% RSLogix 500 project InventoryManagement.RSS, saved by version 8.30.00.16 %
PROJECT "UNTITLED"    % processor: Bul.1763 MicroLogix 1100 Series B %

PROGRAM FILES
  LAD 2   9 rungs

DATA FILES
  O0 OUTPUT  4 elements
  I1 INPUT  6 elements
  S2 STATUS  66 elements
  B3 BINARY  1 elements
  T4 TIMER  1 elements
  C5 COUNTER  1 elements
  R6 CONTROL  1 elements
  N7 INTEGER  11 elements
  F8 FLOAT  1 elements
  ST9 STRING  10 elements

LADDER 2
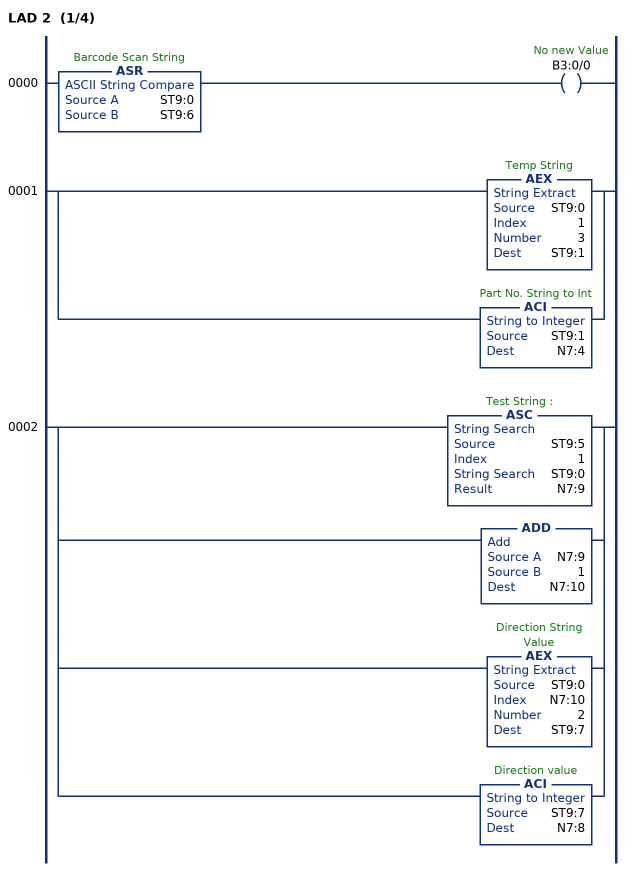
% Rung: 0 %
SOR ASR ST9:0 ST9:6 OTE B3:0/0 EOR
%   ST9:0  "Barcode Scan String" %
%   B3:0/0  "No new Value" %
% Rung: 1 %
SOR BST AEX ST9:0 1 3 ST9:1 NXB ACI ST9:1 N7:4 BND EOR
%   ST9:0  "Barcode Scan String" %
%   ST9:1  "Temp String" %
%   N7:4  "Part No. String to Int" %
% Rung: 2 %
SOR BST ASC ST9:5 1 ST9:0 N7:9 NXB ADD N7:9 1 N7:10 NXB AEX ST9:0 N7:10 2 ST9:7 NXB ACI ST9:7 N7:8 BND EOR
%   ST9:5  "Test String :" %
%   ST9:0  "Barcode Scan String" %
%   ST9:7  "Direction String Value" %
%   N7:8  "Direction value" %

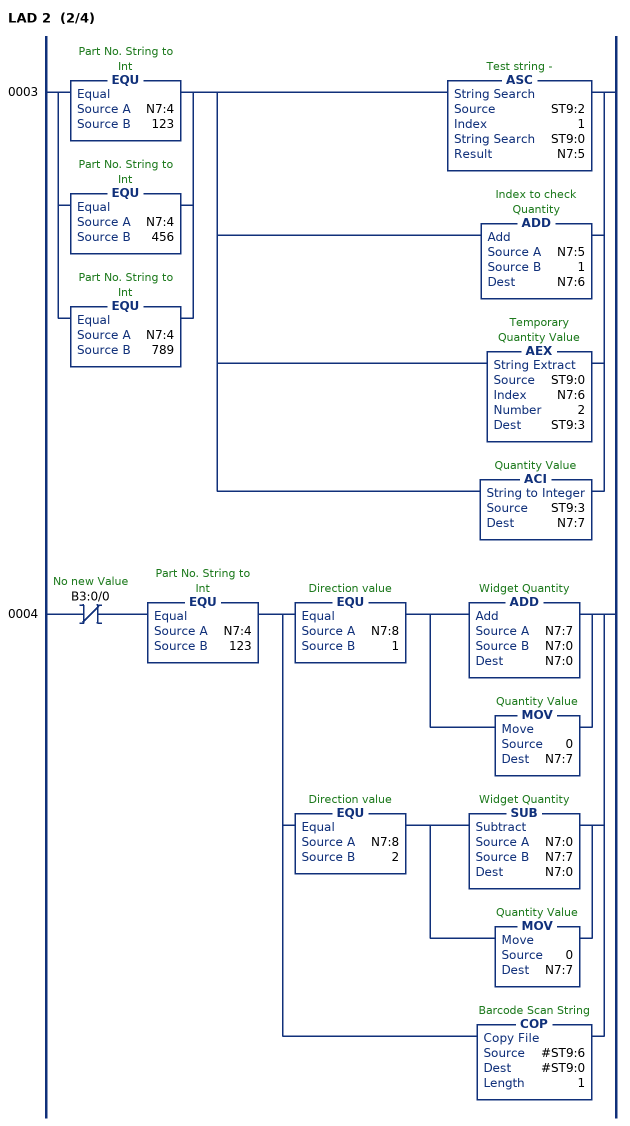
% Rung: 3 %
SOR BST EQU N7:4 123 NXB EQU N7:4 456 NXB EQU N7:4 789 BND BST ASC ST9:2 1 ST9:0 N7:5 NXB ADD N7:5 1 N7:6 NXB AEX ST9:0 N7:6 2 ST9:3 NXB ACI ST9:3 N7:7 BND EOR
%   N7:4  "Part No. String to Int" %
%   ST9:2  "Test string -" %
%   ST9:0  "Barcode Scan String" %
%   N7:5  "Target Start Index" %
%   N7:6  "Index to check Quantity" %
%   ST9:3  "Temporary Quantity Value" %
%   N7:7  "Quantity Value" %
% Rung: 4 %
SOR XIO B3:0/0 EQU N7:4 123 BST EQU N7:8 1 BST ADD N7:7 N7:0 N7:0 NXB MOV 0 N7:7 BND NXB EQU N7:8 2 BST SUB N7:0 N7:7 N7:0 NXB MOV 0 N7:7 BND NXB COP #ST9:6 #ST9:0 1 BND EOR
%   B3:0/0  "No new Value" %
%   N7:4  "Part No. String to Int" %
%   N7:8  "Direction value" %
%   N7:7  "Quantity Value" %
%   N7:0  "Widget Quantity" %
%   ST9:0  "Barcode Scan String" %

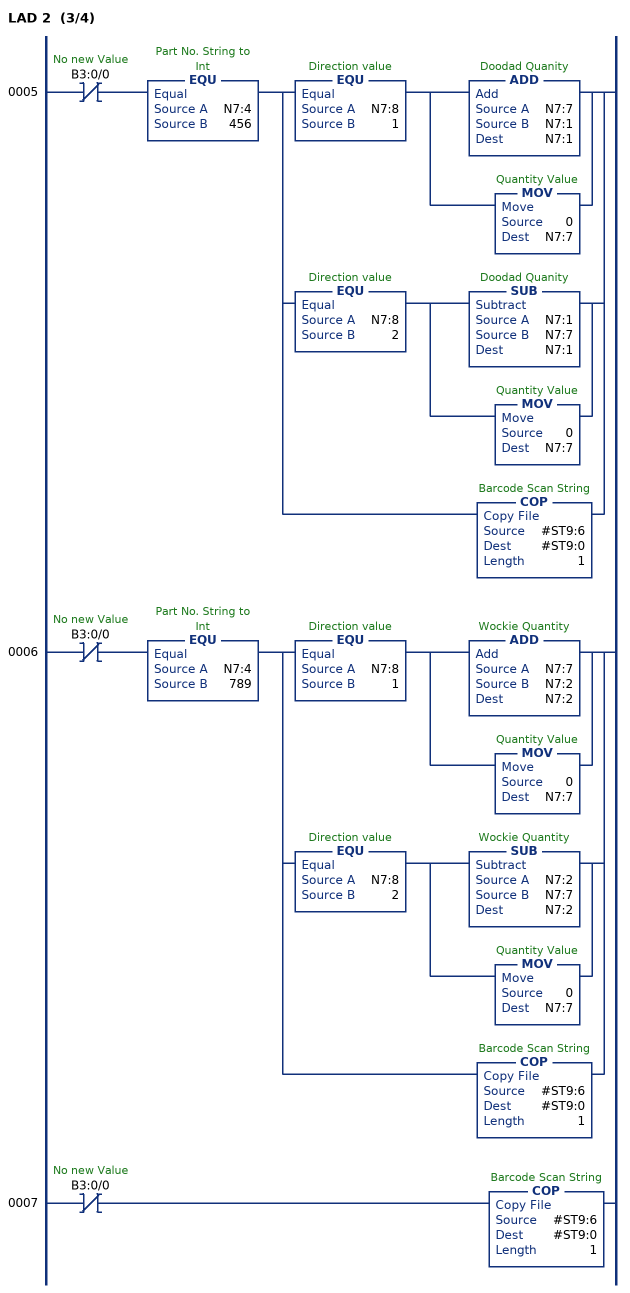
% Rung: 5 %
SOR XIO B3:0/0 EQU N7:4 456 BST EQU N7:8 1 BST ADD N7:7 N7:1 N7:1 NXB MOV 0 N7:7 BND NXB EQU N7:8 2 BST SUB N7:1 N7:7 N7:1 NXB MOV 0 N7:7 BND NXB COP #ST9:6 #ST9:0 1 BND EOR
%   B3:0/0  "No new Value" %
%   N7:4  "Part No. String to Int" %
%   N7:8  "Direction value" %
%   N7:7  "Quantity Value" %
%   N7:1  "Doodad Quanity" %
%   ST9:0  "Barcode Scan String" %
% Rung: 6 %
SOR XIO B3:0/0 EQU N7:4 789 BST EQU N7:8 1 BST ADD N7:7 N7:2 N7:2 NXB MOV 0 N7:7 BND NXB EQU N7:8 2 BST SUB N7:2 N7:7 N7:2 NXB MOV 0 N7:7 BND NXB COP #ST9:6 #ST9:0 1 BND EOR
%   B3:0/0  "No new Value" %
%   N7:4  "Part No. String to Int" %
%   N7:8  "Direction value" %
%   N7:7  "Quantity Value" %
%   N7:2  "Wockie Quantity" %
%   ST9:0  "Barcode Scan String" %
% Rung: 7 %
SOR XIO B3:0/0 COP #ST9:6 #ST9:0 1 EOR
%   B3:0/0  "No new Value" %
%   ST9:0  "Barcode Scan String" %

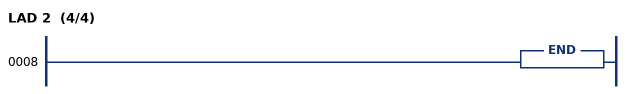
% Rung: 8 %
SOR END EOR

OTHER DOCUMENTED ADDRESSES
  B3:0/1  "ONS"
  B3:0/2  "ONS"
  B3:0/3  "ONS"
  ST9:4  "Temporary Direction String"
  ST9:5.0  "Test String"
  ST9:6.0  "Move empty string to source"

DATA TABLE (non-zero values as saved)
DATA N7
% N7:0 % 1 1 1 0 149 4 5 29 1 6
% N7:10 % 7
DATA ST9
% ST9:1 % "124"
% ST9:2 % "-"
% ST9:3 % "10"
% ST9:5 % ":"
% ST9:7 % "1"
